FUNCTION_BLOCK FB_VPC EXTENDS FB_CtrlBase
VAR_INPUT
	In_bolVacuumOk			: BOOL;
	In_bolPumpOk			: BOOL;
END_VAR
VAR_OUTPUT
	Out_bolVaccumPumpOn		: BOOL;
END_VAR
VAR
	/// Specific interface struct for public access
	SIf					: T_Ctrl_SIf_VPC;
END_VAR

(*__________________________________________________________________________________________________
¦	
¦	Vistaprint Schweiz GmbH
¦	CH - 8401 Winterthur
¦
¦	www.vistaprint.ch - info@vistaprint.ch
¦___________________________________________________________________________________________________

Function desription:
Vacuum Pump implementation. 


History:
Version		Date			Author		Comment
---------------------------------------------------------------------------------------------------
0.00.1		09.07.2013		PC			Start history
___________________________________________________________________________________________________*)


SUPER^();

(*
IF (me.bolActivate) THEN // cyclic call enabled
	IF (CIf.Info.bolInitDone=FALSE) THEN // first cycle -> init
		CtrlInit();
		CIf.Info.bolInitDone := TRUE;
	ELSE
		CycleStartDuty();
	
		Always();
		
		StateMachine();
		
		CycleEndDuty();
	END_IF
END_IF;
*)

METHOD PROTECTED sta_RUNBusy : BOOL
VAR_INPUT
END_VAR
// state implemetation
//--------------------------------------------------------------------------------------
// Entry action
	IF (me.StateMachine.intState<>me.StateMachine.intStateLastCycle) THEN
		me.StateMachine.intStateLastCycle := me.StateMachine.intState;
		SIf.Out.bolVacuumPumpOn.intern := TRUE;

		fbSimulationTimer.IN := FALSE;
		fbSimulationTimer.PT := UDINT_TO_TIME(SIf.Par.udiSimVacuumPumpOnTime_ms);
		fbSimulationTimer(); // set time/reset timer
		fbSimulationTimer.IN := TRUE; // start timer
	END_IF


//--------------------------------------------------------------------------------------
// Cyclic action
	IF (me.StateMachine.intState=me.StateMachine.intStateLastCycle) THEN
		// Simulation
		IF (CIf.SwCfg.bolSimulation) THEN
			fbSimulationTimer(); // simulation time
			IF (fbSimulationTimer.Q) THEN
				SIf.In.bolPumpOn.intern := TRUE;
				SIf.In.bolVacuumOk.intern := TRUE;
			END_IF
		END_IF

		IF ((SIf.In.bolVacuumOk.intern) OR (NOT SIf.Cfg.VacuumPumpFeedback)) AND ((SIf.In.bolVacuumOk.intern) OR (NOT SIf.Cfg.VacuumSensorAvailable)) THEN
			me.StateMachine.intStateNext := VPC_CmdState.cSTA_VPC_StabilizeBusy;
		END_IF;		
		
		IF (me.StateMachine.udiTimeInState_ms > SIf.Par.udiVacuumPumpTime_ms) THEN
			IF (NOT SIf.In.bolPumpOn.intern) AND (SIf.Cfg.VacuumPumpFeedback) THEN
				pfbAlarmCtrl^.setAlarm(CIf.Info.intCtrlId,INT_TO_UINT(E_ALM_VPC.VacuumPumpOnTimeout),0,ADR(SIf.Alm),E_AlmState.RST,CIf.Job.eMe_ActivAlmClass);
			END_IF;

			IF ((NOT SIf.In.bolVacuumOk.intern) AND (SIf.Cfg.VacuumSensorAvailable)) THEN
				pfbAlarmCtrl^.setAlarm(CIf.Info.intCtrlId,INT_TO_UINT(E_ALM_VPC.VacuumFailure),0,ADR(SIf.Alm),E_AlmState.RST,CIf.Job.eMe_ActivAlmClass);
			END_IF;	

			me.StateMachine.intStateNext :=  cSTA_ERROR;
		END_IF
	END_IF


//--------------------------------------------------------------------------------------
// Exit action
	IF (me.StateMachine.intState<>me.StateMachine.intStateNext) THEN
		;
	END_IF
END_METHOD

METHOD PROTECTED IoOutBridge : BOOL
VAR
	bolSwitchValvesOff: BOOL;
END_VAR
// digitale and analoge inputs read from hardware or forcing
IF (CIf.SwCfg.bolSimulation = FALSE) THEN
	setOutBol(CIf.Job.bolIoForce ,ADR(SIf.Out.bolVacuumPumpOn));

	THIS^.Out_bolVaccumPumpOn := SIf.Out.bolVacuumPumpOn.map;
END_IF
END_METHOD

METHOD getCtrlSIf : POINTER TO T_Ctrl_SIf_VPC
getCtrlSIf := ADR(SIf);
END_METHOD

METHOD FB_init : BOOL
VAR_INPUT
	bInitRetains : BOOL; // if TRUE, the retain variables are initialized (warm start / cold start)
	bInCopyCode : BOOL;  // if TRUE, the instance afterwards gets moved into the copy code (online change)
END_VAR
VAR
	iIdx		: UINT;
	iLength		: UINT;	
END_VAR
//------------------------------------------------------------------------------------------------------------------------
// to manually change in new FUB implementation!!!
// define valid commands for this controller
iLength := SIZEOF(CIf.Job.aCmdList)/SIZEOF(CIf.Job.aCmdList[0]);
iIdx := 0;

WHILE (iIdx < iLength) AND (CIf.Job.aCmdList[iIdx].intCmd <> cCMD_INITIALIZED) DO
	iIdx := iIdx + 1; 
END_WHILE

IF (iIdx < iLength) THEN
// Add configuration of own comands	
	CIf.Job.aCmdList[iIdx].intCmd := BASE_PLC.cCMD_RUN;
	CIf.Job.aCmdList[iIdx].strName := 'RUN'; 
	CIf.Job.aCmdList[iIdx].bolAvailable := TRUE;
ELSE
	// Error if the aCmdList Array is to small
END_IF

// set name of class/typ
CIf.Info.strType := 'FB_VPC';
CIf.Info.strFullName := 'Vacuum Pump Controller';

// set alarm class
SIf.Alm[E_ALM_VPC.VacuumPumpOnTimeout].eAlmClass := E_AlmClass.TSTOP;
SIf.Alm[E_ALM_VPC.VacuumPumpOnTimeout].strText := 'Vacuum pump On timeout'; 
SIf.Alm[E_ALM_VPC.VacuumPumpOffTimeout].eAlmClass := E_AlmClass.TSTOP;
SIf.Alm[E_ALM_VPC.VacuumPumpOffTimeout].strText := 'Vacuum pump Off timeout';
SIf.Alm[E_ALM_VPC.VacuumFailure].eAlmClass := E_AlmClass.TSTOP;
SIf.Alm[E_ALM_VPC.VacuumFailure].strText := 'Vacuum failure';

//*******************************************************************************
// initial values
//*******************************************************************************

// software configuration
CIf.SwCfg.bolExist := TRUE;
CIf.SwCfg.bolEnable := TRUE;
CIf.SwCfg.bolSimulation := FALSE;

// parameter
SIf.Par.udiVacuumPumpTime_ms := 10000;
SIf.Par.udiVacuumStabilizationTime_ms := 3000;
SIf.Par.udiSimVacuumPumpOnTime_ms := SIf.Par.udiVacuumPumpTime_ms / 2;
END_METHOD

METHOD PROTECTED Always : BOOL
SUPER^.Always();

// ----------------------------------------------------------------------------------
// cyclic actions outside of statemachine
IF (me.StateMachine.intState<>cSTA_SINGLE_ANSWER) THEN
	
	; // always error supervision
	
END_IF

// ----------------------------------------------------------------------------------
// Conditions Always
IF (((me.Alarm.eActivAlmClass=E_AlmClass.EOFF) OR (me.Alarm.eActivAlmClass=E_AlmClass.OFF) OR (me.intCmd=cCMD_OFF))
		 AND (me.StateMachine.intState<>cSTA_ERROR) AND (me.StateMachine.intState<>cSTA_ERRORQuit) AND
		(me.StateMachine.intState<>cSTA_OFF) AND (me.StateMachine.intState<>cSTA_OFFBusy)) THEN
	// alarm evt EOFF, OFF or cmd off
	me.StateMachine.intStateNext := cSTA_OFFBusy;
END_IF
END_METHOD

METHOD PROTECTED sta_StabilizeVacuum : BOOL
VAR_INPUT
END_VAR
// state implemetation
//--------------------------------------------------------------------------------------
// Entry action
	IF (me.StateMachine.intState<>me.StateMachine.intStateLastCycle) THEN
		me.StateMachine.intStateLastCycle := me.StateMachine.intState;
	END_IF


//--------------------------------------------------------------------------------------
// Cyclic action
	IF (me.StateMachine.intState=me.StateMachine.intStateLastCycle) THEN
		// State Change Condition
		
		IF (me.StateMachine.udiTimeInState_ms > SIf.Par.udiVacuumStabilizationTime_ms) THEN
			me.StateMachine.intStateNext :=  BASE_PLC.cSTA_RUN;
		END_IF;	

		IF (NOT SIf.In.bolPumpOn.intern) AND (SIf.Cfg.VacuumPumpFeedback) THEN
			pfbAlarmCtrl^.setAlarm(CIf.Info.intCtrlId,INT_TO_UINT(E_ALM_VPC.VacuumPumpOnTimeout),0,ADR(SIf.Alm),E_AlmState.RST,CIf.Job.eMe_ActivAlmClass);
			me.StateMachine.intStateNext :=  BASE_PLC.cSTA_ERROR;
		END_IF;

		IF ((NOT SIf.In.bolVacuumOk.intern) AND (SIf.Cfg.VacuumSensorAvailable)) THEN
			pfbAlarmCtrl^.setAlarm(CIf.Info.intCtrlId,INT_TO_UINT(E_ALM_VPC.VacuumFailure),0,ADR(SIf.Alm),E_AlmState.RST,CIf.Job.eMe_ActivAlmClass);
			me.StateMachine.intStateNext :=  BASE_PLC.cSTA_ERROR;
		END_IF;	
	END_IF


//--------------------------------------------------------------------------------------
// Exit action
	IF (me.StateMachine.intState<>me.StateMachine.intStateNext) THEN
		;
	END_IF
END_METHOD

METHOD PROTECTED sta_OFFBusy : BOOL
VAR_INPUT
END_VAR
// state implemetation
//--------------------------------------------------------------------------------------
// Entry action
	IF (me.StateMachine.intState<>me.StateMachine.intStateLastCycle) THEN
		me.StateMachine.intStateLastCycle := me.StateMachine.intState;
		// Switch Pump Off
		SIf.Out.bolVacuumPumpOn.intern := FALSE;
	END_IF


//--------------------------------------------------------------------------------------
// Cyclic action
	IF (me.StateMachine.intState=me.StateMachine.intStateLastCycle) THEN
		IF (CIf.SwCfg.bolSimulation) THEN
			SIf.In.bolPumpOn.intern := FALSE;
			SIf.In.bolVacuumOk.intern := FALSE;
		END_IF

		IF ((NOT SIf.In.bolPumpOn.intern) OR (NOT SIf.Cfg.VacuumPumpFeedback)) AND ((NOT SIf.In.bolVacuumOk.intern) OR (NOT SIf.Cfg.VacuumSensorAvailable)) THEN
			me.StateMachine.intStateNext := BASE_PLC.cSTA_OFF;
		END_IF;	
	END_IF


//--------------------------------------------------------------------------------------
// Exit action
	IF (me.StateMachine.intState<>me.StateMachine.intStateNext) THEN
		;
	END_IF
END_METHOD

METHOD PROTECTED sta_OFF : BOOL
VAR_INPUT
END_VAR
// state implemetation
//--------------------------------------------------------------------------------------
// Entry action
	IF (me.StateMachine.intState<>me.StateMachine.intStateLastCycle) THEN
		me.StateMachine.intStateLastCycle := me.StateMachine.intState;

	END_IF


//--------------------------------------------------------------------------------------
// Cyclic action
	IF (me.StateMachine.intState=me.StateMachine.intStateLastCycle) THEN
		IF me.intCmd = BASE_PLC.cCMD_RUN THEN
			me.StateMachine.intStateNext := BASE_PLC.cSTA_RUNBusy;
		END_IF
	END_IF


//--------------------------------------------------------------------------------------
// Exit action
	IF (me.StateMachine.intState<>me.StateMachine.intStateNext) THEN
		;
	END_IF
END_METHOD

METHOD PROTECTED getCmdState : STRING

VAR_INPUT
	intCmdState: INT;
	bolState: BOOL;
END_VAR
getCmdState := SUPER^.getCmdState(intCmdState:=intCmdState,bolState:=bolState); // get global/base defined cmds/states

IF (getCmdState='') THEN // global not defined get local
	// get string cmd/state string information in runtime
	IF (bolState=FALSE) THEN
		;// Comands's
	ELSE
		// States's
		CASE intCmdState OF
			VPC_CmdState.cSTA_VPC_StabilizeBusy: 
				getCmdState := 'cSTA_StabilizeBusy';
		END_CASE;
	END_IF
END_IF
END_METHOD

METHOD PROTECTED sta_RUN : BOOL
VAR_INPUT
END_VAR
// state implemetation
//--------------------------------------------------------------------------------------
// Entry action
	IF (me.StateMachine.intState<>me.StateMachine.intStateLastCycle) THEN
		me.StateMachine.intStateLastCycle := me.StateMachine.intState;
	END_IF


//--------------------------------------------------------------------------------------
// Cyclic action
	IF (me.StateMachine.intState=me.StateMachine.intStateLastCycle) THEN
		// State Change Condition
		IF (NOT SIf.In.bolPumpOn.intern) AND (SIf.Cfg.VacuumPumpFeedback) THEN
			pfbAlarmCtrl^.setAlarm(CIf.Info.intCtrlId,INT_TO_UINT(E_ALM_VPC.VacuumPumpOnTimeout),0,ADR(SIf.Alm),E_AlmState.RST,CIf.Job.eMe_ActivAlmClass);
			me.StateMachine.intStateNext :=  BASE_PLC.cSTA_ERROR;
		END_IF;

		IF ((NOT SIf.In.bolVacuumOk.intern) AND (SIf.Cfg.VacuumSensorAvailable)) THEN
			pfbAlarmCtrl^.setAlarm(CIf.Info.intCtrlId,INT_TO_UINT(E_ALM_VPC.VacuumFailure),0,ADR(SIf.Alm),E_AlmState.RST,CIf.Job.eMe_ActivAlmClass);
			me.StateMachine.intStateNext :=  BASE_PLC.cSTA_ERROR;
		END_IF;	
	END_IF


//--------------------------------------------------------------------------------------
// Exit action
	IF (me.StateMachine.intState<>me.StateMachine.intStateNext) THEN
		;
	END_IF
END_METHOD

METHOD PROTECTED sta_PON : BOOL
VAR_INPUT
END_VAR
// state implemetation
//--------------------------------------------------------------------------------------
// Entry action
	IF (me.StateMachine.intState<>me.StateMachine.intStateLastCycle) THEN
		me.StateMachine.intStateLastCycle := me.StateMachine.intState;
		
	END_IF


//--------------------------------------------------------------------------------------
// Cyclic action
	IF (me.StateMachine.intState=me.StateMachine.intStateLastCycle) THEN
		;
	END_IF




//--------------------------------------------------------------------------------------
// Exit action
	IF (me.StateMachine.intState<>me.StateMachine.intStateNext) THEN
		;
	END_IF
END_METHOD

METHOD PROTECTED sta_ERROR : BOOL
// state implemetation
//--------------------------------------------------------------------------------------
// Entry action
	IF (me.StateMachine.intState<>me.StateMachine.intStateLastCycle) THEN
		me.StateMachine.intStateHistory := me.StateMachine.intStateLastCycle; // -> possibillity to go back to state before error
		me.StateMachine.intStateLastCycle := me.StateMachine.intState;
		
	END_IF


//--------------------------------------------------------------------------------------
// Cyclic action
	IF (me.StateMachine.intState=me.StateMachine.intStateLastCycle) THEN
		
		;
		
		
		// State Change Condition
		IF (CIf.Job.bolAlmReset = TRUE) THEN
			me.StateMachine.intStateNext := cSTA_ERRORQuit;
		END_IF
	END_IF




//--------------------------------------------------------------------------------------
// Exit action
	IF (me.StateMachine.intState<>me.StateMachine.intStateNext) THEN
		;
	END_IF
END_METHOD

METHOD PROTECTED IoInBridge : BOOL
// digitale and analoge inputs read from hardware or forcing
SIf.In.bolVacuumOk.map := THIS^.In_bolVacuumOk;
SIf.In.bolPumpOn.map := THIS^.In_bolPumpOk;

IF (CIf.SwCfg.bolSimulation = FALSE) THEN
	getInBol(CIf.Job.bolIoForce,ADR(SIf.In.bolVacuumOk));
	getInBol(CIf.Job.bolIoForce,ADR(SIf.In.bolPumpOn));
ELSE
	//simulation of global IO
END_IF
END_METHOD

METHOD PROTECTED StateMachine : BOOL
SUPER^.StateMachine();

// main statemachine of base controller
CASE me.StateMachine.intState OF
    VPC_CmdState.cSTA_VPC_StabilizeBusy: 
        THIS^.sta_StabilizeVacuum();
	cSTA_RUNBusy: 
        THIS^.sta_RUNBusy();
    cSTA_RUN: 
        THIS^.sta_RUN();
END_CASE;
END_METHOD

METHOD PROTECTED sta_ERRORQuit : BOOL
// state implemetation
//--------------------------------------------------------------------------------------
// Entry action
	IF (me.StateMachine.intState<>me.StateMachine.intStateLastCycle) THEN
		me.StateMachine.intStateLastCycle := me.StateMachine.intState;
		
	END_IF


//--------------------------------------------------------------------------------------
// Cyclic action
	IF (me.StateMachine.intState=me.StateMachine.intStateLastCycle) THEN
		
		;
		// evtl. wait time if reset of device is necessary and then decide to go to states or ERROR state
		IF (CIf.Job.bolAlmReset = TRUE) THEN
			CIf.Job.eMe_ActivAlmClass := E_AlmClass.NONE; // reset feedback channel for parent
			CIf.Job.bolAlmReset := FALSE;
		END_IF
		
		// State Change Condition
		IF (CIf.Job.bolAlmReset = FALSE) THEN
			IF (me.StateMachine.intStateHistory<=cSTA_PON) THEN
				me.StateMachine.intStateNext := cSTA_PONBusy;
			ELSIF(me.intCmd=cCMD_OFF) THEN
				me.StateMachine.intStateNext := cSTA_OFFBusy;
			ELSIF(me.intCmd=cCMD_STOP) THEN
				me.StateMachine.intStateNext := cSTA_STOPBusy;
			ELSIF(me.intCmd=BASE_PLC.cCMD_RUN) THEN
				me.StateMachine.intStateNext := BASE_PLC.cSTA_RUNBusy;
			END_IF
		END_IF
	END_IF




//--------------------------------------------------------------------------------------
// Exit action
	IF (me.StateMachine.intState<>me.StateMachine.intStateNext) THEN
		;
	END_IF
END_METHOD

END_FUNCTION_BLOCK

(* stored: Version 1.1.0.1, ProductVersion 3.1.0.25
   POU FB_VPC: Id {13511828-5fa3-4db9-8a62-883d17247bf0}
   Method sta_RUNBusy: Id {1597373b-6e96-49e1-bdbf-9fa98235040c}
   Method IoOutBridge: Id {3b060d29-e9cf-457f-8c49-0301ccd0cca5}
   Method getCtrlSIf: Id {3f73b4c8-fe1a-4e64-b16a-7e0063e5c6aa}
   Method FB_init: Id {49182cc1-4f51-4fb4-9202-ff24f518710e}
   Method Always: Id {4f56d2f9-8407-4812-8ceb-f4f26f794649}
   Method sta_StabilizeVacuum: Id {56e99b8a-45db-4a94-b998-af0d9227c626}
   Method sta_OFFBusy: Id {58e778f2-58e2-4242-b691-65410b4a0daa}
   Method sta_OFF: Id {69e589e4-f383-473e-b644-e3226d6d511f}
   Method getCmdState: Id {703f6dd4-8675-4294-8b3d-2f6ff473bc8c}
   Method sta_RUN: Id {814d30da-f6f2-44a3-8f69-fbdc9cbd5a0a}
   Method sta_PON: Id {cd944ca7-9f97-4fb3-b4a2-4d1ad61c9f19}
   Method sta_ERROR: Id {cdcdfbea-0d76-4965-a714-0ee8fc61cf6a}
   Method IoInBridge: Id {e901586d-7f23-48a3-af3c-72b64ab38fc4}
   Method StateMachine: Id {fb3e697c-bec3-4662-ad64-257ff20479d8}
   Method sta_ERRORQuit: Id {fbdec985-78a5-46c9-a569-cae78f6ce0ca} *)
